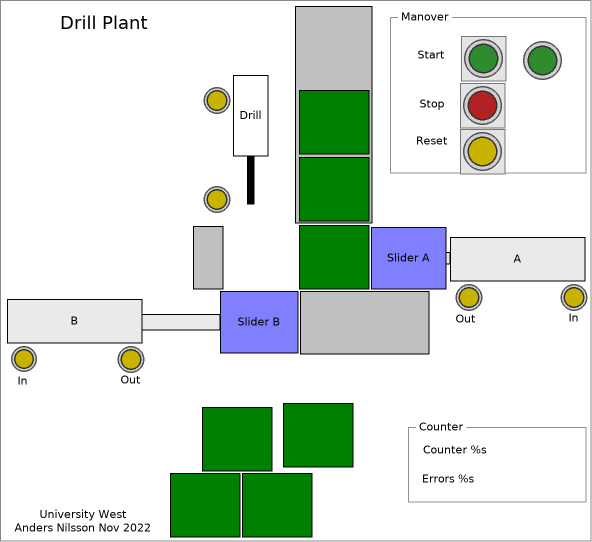
VISUALIZATION Visualization  // 592x542
    Group (233,75 59x138)
        p2773130477: main.nPosDrill
        p1126004900: MAIN.nPosDrill
        Rectangle (0,0 35x81), "Drill"
        Rectangle (14,81 7x48)
    Rectangle (295,6 77x217)
    Rectangle (299,225 70x64), invisible if: MAIN.mxCubeInvisible
        p3528305787: MAIN.nPosXCube
        p874137650: MAIN.nPosXCube
        p2773130477: MAIN.nPosYCube
        p1126004900: MAIN.nPosYCube
    Rectangle (193,226 30x63)
    Rectangle (299,157 70x64)
    Rectangle (300,291 129x63)
    Rectangle (299,90 70x64)
    Lamp1 (115,344 32x31), variable: MAIN.qxSliderBout, style: Lamp-Lamp1-Yellow
    Lamp1 (8,344 32x30), variable: MAIN.qxSliderBin, style: Lamp-Lamp1-Yellow
    Lamp1 (558,282 32x31), variable: MAIN.qxSliderAin, style: Lamp-Lamp1-Yellow
    Lamp1 (453,282 32x31), variable: MAIN.qxSliderAout, style: Lamp-Lamp1-Yellow
    Lamp1 (201,85 32x31), variable: MAIN.qxDrillUp, style: Lamp-Lamp1-Yellow
    Lamp1 (201,184 32x31), variable: MAIN.qxDrillDown, style: Lamp-Lamp1-Yellow
    Rectangle (242,473 70x64), invisible if: main.nCnt < 1
    Rectangle (283,403 70x64), invisible if: main.nCnt < 4
    Rectangle (170,473 70x64), invisible if: main.nCnt < 2
    Rectangle (202,407 70x64), invisible if: main.nCnt < 3
    GroupBox (390,9 196x164), "Manover"
        Label (20,23 42x46), "Start"
        PushSwitch (71,27 45x45), variable: MAIN.qxButtonStart, behaviour: TAP, style: Switch-PushSwitch-Green
        PushSwitch (70,74 45x45), variable: MAIN.qxButtonStop, behaviour: TAP, style: Switch-PushSwitch-Red
        Lamp1 (130,29 45x45), variable: MAIN.ixLampStarted, style: Lamp-Lamp1-Green
        Label (21,72 42x46), "Stop"
        PushSwitch (70,120 45x45), variable: MAIN.mxReset, behaviour: TAP, style: Switch-PushSwitch-Yellow
    GroupBox (408,419 178x83), "Counter"
        Rectangle (12,16 112x30), "Counter %s", text variable: MAIN.nCnt
        Rectangle (11,45 112x30), "Errors %s", text variable: MAIN.nErrorCnt
    Label (447,302 37x34), "Out"
    Label (112,363 37x34), "Out"
    Label (555,301 37x34), "In"
    Label (4,364 37x34), "In"
    Label (411,118 42x46), "Reset"
    Rectangle (371,252 79x12)
    Rectangle (450,237 135x44), "A"
    Rectangle (139,314 81x16)
    Rectangle (7,299 135x44), "B"
    Rectangle (371,227 75x62), "Slider A"
        p3528305787: MAIN.nPosSliderA
        p874137650: MAIN.nPosSliderA
    Rectangle (220,291 78x62), "Slider B"
        p3528305787: MAIN.nPosSliderB
        p874137650: MAIN.nPosSliderB
    Label (26,6 156x34), "Drill Plant"
    Label (7,500 152x42), "University West Anders Nilsson Nov 2022"
END_VISUALIZATION

(* stored: Version 1.1.0.1, ProductVersion 3.1.4024.11
   Visu Visualization: Id {6a967cc4-b88c-4500-a7a1-abfc74b431c0} *)
